// TIA Portal V18 export
TYPE "MEStoPLC_AGVExchange"
// stored: IsFailsafeCompliant false
   STRUCT
      "M-PosCallDone1" : Byte;   // AGV站点1呼叫完成（MES） 1-已呼叫 2-呼叫异常 设备将对应的呼叫信号一起复位
      "M-PosCallDone2" : Byte;   // AGV站点2呼叫完成（MES） 1-已呼叫 2-呼叫异常 设备将对应的呼叫信号一起复位
      "M-PosCallDone3" : Byte;   // AGV站点3呼叫完成（MES） 1-已呼叫 2-呼叫异常 设备将对应的呼叫信号一起复位
      "M-PosCallDone4" : Byte;   // AGV站点4呼叫完成（MES） 1-已呼叫 2-呼叫异常 设备将对应的呼叫信号一起复位
      "M-PosCallDone5" : Byte;   // AGV站点4呼叫完成（MES） 1-已呼叫 2-呼叫异常 设备将对应的呼叫信号一起复位
      Reserve : Array[1..994] of Byte;   // AGV交互预留
   END_STRUCT;
END_TYPE
